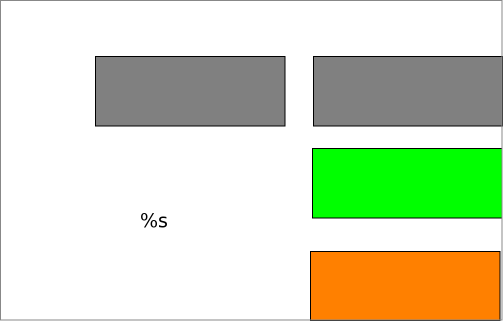
VISUALIZATION AnimCRAH  // 503x321
VAR_INPUT
	idCrah : WSTRING;
	Offline : BOOL;
	Alarm : BOOL;
	Enable : BOOL;
	Running : BOOL;
	Inhibited : BOOL;
	Maintenance : BOOL;
	HOA : WORD;
	Isolator1 : BOOL;
	Isolator2 : BOOL;
	DeactivateIso2 : BOOL;
END_VAR
    Rectangle (95,56 190x70), colour toggle: Enable
    Rectangle (313,56 190x70), colour toggle: Enable
    Rectangle (79,206 150x30), "%s", text list: 'CRAH_Status', text index: HOA
    Rectangle (312,148 190x70), colour toggle: Enable, invisible if: not Running
    Rectangle (310,251 190x70), colour toggle: Enable, invisible if: not Inhibited
END_VISUALIZATION

(* stored: Version 1.1.0.1, ProductVersion 3.1.4024.12
   Visu AnimCRAH: Id {0c9e31ed-12e5-4609-bc03-d7b967d3918f} *)
